// TIA Portal V19 export
FUNCTION_BLOCK "Area02_SafetyInterface_FB"   // FB207, LAD
TITLE = AREA 01 SAFETY INTERFACE
// stored: Access Published, MemoryReserve 100, SetENOAutomatically false
   VAR_INPUT
      AreaInterface : "AreaInterface";
      Passivation : Bool;
   END_VAR
   VAR_OUTPUT
      MachineInterface : "MachineInterface";
      COut : Struct
         WarningsPresence : Bool;
         AlarmsPresence : Bool;
         PathTestRollformer_DriveCtrlSafe : Bool;
      END_STRUCT;
   END_VAR
   VAR_IN_OUT
      Alarm : Struct
         FDBACK_Error : Struct
            F_Contactor_Rollformer_CambioFormato : Bool;
            F_Contactor_FinalCut_HU_Motor : Bool;
            F_Contactor_FinalCut_HU_Valve : Bool;
         END_STRUCT;
         S120_SafetyFaultActive : Struct
            Cassetta1_OP : Bool;
            Cassetta1_MOT : Bool;
            Cassetta2_OP : Bool;
            Cassetta2_MOT : Bool;
            Cassetta3_OP : Bool;
            Cassetta3_MOT : Bool;
            Rollformer : Bool;
            FAK_PusherAx : Bool;
            FlyCarriage : Bool;
            AccRolls1 : Bool;
            AccRolls2 : Bool;
            AccRolls3 : Bool;
         END_STRUCT;
         UnathorizedOpen : Struct
            D10 : Bool;
            D11 : Bool;
            D12 : Bool;
            D14 : Bool;
            D15 : Bool;
            D16 : Bool;
            D18 : Bool;
         END_STRUCT;
         PathTest_Rollformer : Bool;
      END_STRUCT;
      Warning : Struct
         Selectors : Struct
            Maintenance_MB2 : Bool;
         END_STRUCT;
         Feedback : Struct
            F_Valve_Area02_HU : Bool;
         END_STRUCT;
         DoorOpened : Struct
            D10 : Bool;
            D11 : Bool;
            D12 : Bool;
            D14 : Bool;
            D15 : Bool;
            D16 : Bool;
            D18 : Bool;
         END_STRUCT;
         DoorOpenRequest : Struct
            D10 : Bool;
            D11 : Bool;
            D12 : Bool;
            D14 : Bool;
            D15 : Bool;
            D16 : Bool;
            D18 : Bool;
         END_STRUCT;
         PathTest_Rollformer : Bool;
      END_STRUCT;
   END_VAR
   VAR
      Sts : Struct
         FdbackErrorPresence : Bool;
         S120SftyFaultPresence : Bool;
         DoorUnauthorizedOpen : Bool;
         DoorOpened { ExternalAccessible := 'False'; ExternalVisible := 'False'; ExternalWritable := 'False'} : Bool;
         DoorOpenRequest : Bool;
         DoorNotLocked : Bool;
      END_STRUCT;
      PathTest_Rollformer { S7_SetPoint := 'True'} : "PathTest";
   END_VAR
   VAR_TEMP
      SteadyOn : Bool;
      BlinkFast : Bool;
      BlinkLow : Bool;
      DummyLamp : Bool;
   END_VAR
BEGIN

REGION Network 1: <<<< C O N T R O L S A F E T Y D I A G N O S T I C >>>>>
END_REGION

REGION Network 2 (SCL): Fdback error


   #Alarm.FDBACK_Error.F_Contactor_Rollformer_CambioFormato := "Main_Safety_RTG1_DB".F_Zone11.F_Contactor_CambioFormato_Profilatrice.ERROR;
   #Alarm.FDBACK_Error.F_Contactor_FinalCut_HU_Motor := "Main_Safety_RTG1_DB".F_Zone13.F_Contactor_HU_FinalCut_Motor.ERROR;
   #Alarm.FDBACK_Error.F_Contactor_FinalCut_HU_Valve := "Main_Safety_RTG1_DB".F_Zone13.F_SafetyValve_FinalCut.FDO_FBK_ERROR;
END_REGION

REGION Network 3 (SCL): S120 Safety Fault

   #Alarm.S120_SafetyFaultActive.Cassetta1_OP := "Main_Safety_RTG1_DB".F_Zone11.F_Sinamics_Cassetta1_OP.SftyFault;
   #Alarm.S120_SafetyFaultActive.Cassetta1_MOT := "Main_Safety_RTG1_DB".F_Zone11.F_Sinamics_Cassetta1_MOT.SftyFault;
   #Alarm.S120_SafetyFaultActive.Cassetta2_OP := "Main_Safety_RTG1_DB".F_Zone11.F_Sinamics_Cassetta2_OP.SftyFault;
   #Alarm.S120_SafetyFaultActive.Cassetta2_MOT := "Main_Safety_RTG1_DB".F_Zone11.F_Sinamics_Cassetta2_MOT.SftyFault;
   #Alarm.S120_SafetyFaultActive.Cassetta3_OP := "Main_Safety_RTG1_DB".F_Zone11.F_Sinamics_Cassetta3_OP.SftyFault;
   #Alarm.S120_SafetyFaultActive.Cassetta3_MOT := "Main_Safety_RTG1_DB".F_Zone11.F_Sinamics_Cassetta3_MOT.SftyFault;
   #Alarm.S120_SafetyFaultActive.Rollformer := "Main_Safety_RTG1_DB".F_Zone20.F_Sinamics_Rollformer.SftyFault;
   #Alarm.S120_SafetyFaultActive.FAK_PusherAx := "Main_Safety_RTG1_DB".F_Zone13.F_Sinamics_FAK_Pusher.SftyFault;
   #Alarm.S120_SafetyFaultActive.FlyCarriage := "Main_Safety_RTG1_DB".F_Zone13.F_Sinamics_Carriage.SftyFault;
   #Alarm.S120_SafetyFaultActive.AccRolls1 := "Main_Safety_RTG1_DB".F_Zone15.F_Sinamics_AccRolls1.SftyFault;
   #Alarm.S120_SafetyFaultActive.AccRolls2 := "Main_Safety_RTG1_DB".F_Zone15.F_Sinamics_AccRolls2.SftyFault;
   #Alarm.S120_SafetyFaultActive.AccRolls3 := "Main_Safety_RTG1_DB".F_Zone15.F_Sinamics_AccRolls3.SftyFault;
END_REGION

REGION Network 4: Door D10 - Alarm unauthorized door opening
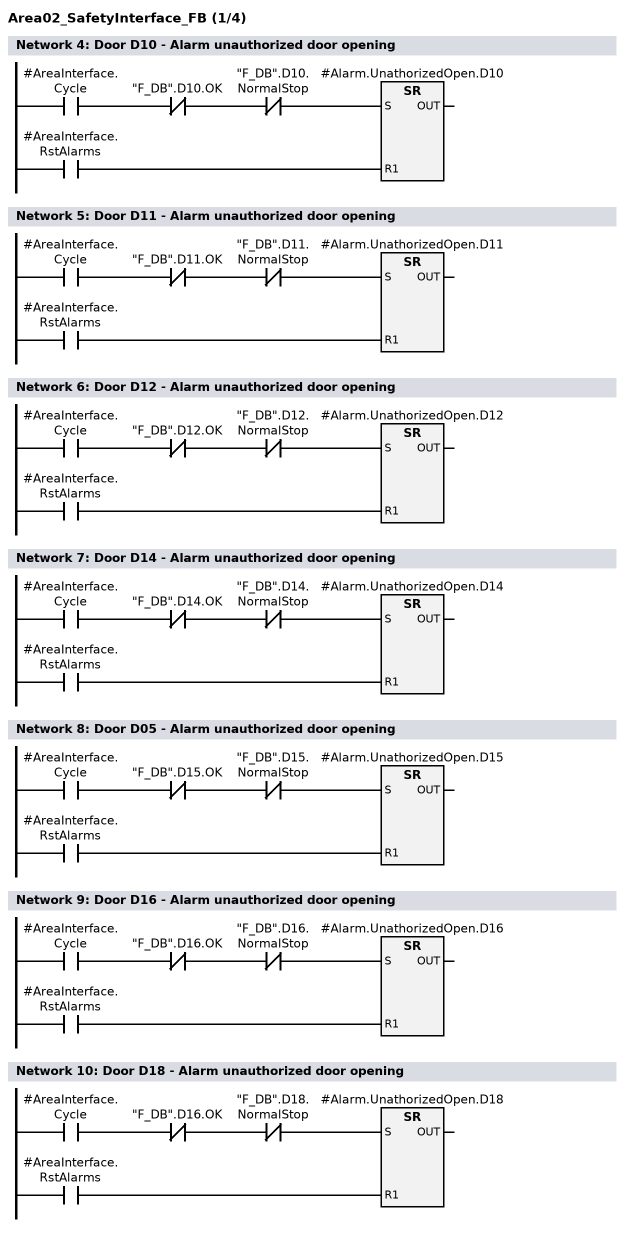
   RUNG wire#powerrail
      Contact( #AreaInterface.Cycle )
      I_Contact( "F_DB".D10.OK )
      I_Contact( "F_DB".D10.NormalStop )
      S_SR(operand := #Alarm.UnathorizedOpen.D10, r1 := wire#w1)
   END_RUNG
   RUNG wire#powerrail
      Contact( #AreaInterface.RstAlarms )
   END_RUNG wire#w1
   // the same network as SCL:
   IF #AreaInterface.Cycle AND NOT "F_DB".D10.OK AND NOT "F_DB".D10.NormalStop THEN
       #Alarm.UnathorizedOpen.D10 := TRUE;   // SR flip-flop
   END_IF;
   IF #AreaInterface.RstAlarms THEN #Alarm.UnathorizedOpen.D10 := FALSE; END_IF;
END_REGION

REGION Network 5: Door D11 - Alarm unauthorized door opening
   RUNG wire#powerrail
      Contact( #AreaInterface.Cycle )
      I_Contact( "F_DB".D11.OK )
      I_Contact( "F_DB".D11.NormalStop )
      S_SR(operand := #Alarm.UnathorizedOpen.D11, r1 := wire#w1)
   END_RUNG
   RUNG wire#powerrail
      Contact( #AreaInterface.RstAlarms )
   END_RUNG wire#w1
   // the same network as SCL:
   IF #AreaInterface.Cycle AND NOT "F_DB".D11.OK AND NOT "F_DB".D11.NormalStop THEN
       #Alarm.UnathorizedOpen.D11 := TRUE;   // SR flip-flop
   END_IF;
   IF #AreaInterface.RstAlarms THEN #Alarm.UnathorizedOpen.D11 := FALSE; END_IF;
END_REGION

REGION Network 6: Door D12 - Alarm unauthorized door opening
   RUNG wire#powerrail
      Contact( #AreaInterface.Cycle )
      I_Contact( "F_DB".D12.OK )
      I_Contact( "F_DB".D12.NormalStop )
      S_SR(operand := #Alarm.UnathorizedOpen.D12, r1 := wire#w1)
   END_RUNG
   RUNG wire#powerrail
      Contact( #AreaInterface.RstAlarms )
   END_RUNG wire#w1
   // the same network as SCL:
   IF #AreaInterface.Cycle AND NOT "F_DB".D12.OK AND NOT "F_DB".D12.NormalStop THEN
       #Alarm.UnathorizedOpen.D12 := TRUE;   // SR flip-flop
   END_IF;
   IF #AreaInterface.RstAlarms THEN #Alarm.UnathorizedOpen.D12 := FALSE; END_IF;
END_REGION

REGION Network 7: Door D14 - Alarm unauthorized door opening
   RUNG wire#powerrail
      Contact( #AreaInterface.Cycle )
      I_Contact( "F_DB".D14.OK )
      I_Contact( "F_DB".D14.NormalStop )
      S_SR(operand := #Alarm.UnathorizedOpen.D14, r1 := wire#w1)
   END_RUNG
   RUNG wire#powerrail
      Contact( #AreaInterface.RstAlarms )
   END_RUNG wire#w1
   // the same network as SCL:
   IF #AreaInterface.Cycle AND NOT "F_DB".D14.OK AND NOT "F_DB".D14.NormalStop THEN
       #Alarm.UnathorizedOpen.D14 := TRUE;   // SR flip-flop
   END_IF;
   IF #AreaInterface.RstAlarms THEN #Alarm.UnathorizedOpen.D14 := FALSE; END_IF;
END_REGION

REGION Network 8: Door D05 - Alarm unauthorized door opening
   RUNG wire#powerrail
      Contact( #AreaInterface.Cycle )
      I_Contact( "F_DB".D15.OK )
      I_Contact( "F_DB".D15.NormalStop )
      S_SR(operand := #Alarm.UnathorizedOpen.D15, r1 := wire#w1)
   END_RUNG
   RUNG wire#powerrail
      Contact( #AreaInterface.RstAlarms )
   END_RUNG wire#w1
   // the same network as SCL:
   IF #AreaInterface.Cycle AND NOT "F_DB".D15.OK AND NOT "F_DB".D15.NormalStop THEN
       #Alarm.UnathorizedOpen.D15 := TRUE;   // SR flip-flop
   END_IF;
   IF #AreaInterface.RstAlarms THEN #Alarm.UnathorizedOpen.D15 := FALSE; END_IF;
END_REGION

REGION Network 9: Door D16 - Alarm unauthorized door opening
   RUNG wire#powerrail
      Contact( #AreaInterface.Cycle )
      I_Contact( "F_DB".D16.OK )
      I_Contact( "F_DB".D16.NormalStop )
      S_SR(operand := #Alarm.UnathorizedOpen.D16, r1 := wire#w1)
   END_RUNG
   RUNG wire#powerrail
      Contact( #AreaInterface.RstAlarms )
   END_RUNG wire#w1
   // the same network as SCL:
   IF #AreaInterface.Cycle AND NOT "F_DB".D16.OK AND NOT "F_DB".D16.NormalStop THEN
       #Alarm.UnathorizedOpen.D16 := TRUE;   // SR flip-flop
   END_IF;
   IF #AreaInterface.RstAlarms THEN #Alarm.UnathorizedOpen.D16 := FALSE; END_IF;
END_REGION

REGION Network 10: Door D18 - Alarm unauthorized door opening
   RUNG wire#powerrail
      Contact( #AreaInterface.Cycle )
      I_Contact( "F_DB".D16.OK )
      I_Contact( "F_DB".D18.NormalStop )
      S_SR(operand := #Alarm.UnathorizedOpen.D18, r1 := wire#w1)
   END_RUNG
   RUNG wire#powerrail
      Contact( #AreaInterface.RstAlarms )
   END_RUNG wire#w1
   // the same network as SCL:
   IF #AreaInterface.Cycle AND NOT "F_DB".D16.OK AND NOT "F_DB".D18.NormalStop THEN
       #Alarm.UnathorizedOpen.D18 := TRUE;   // SR flip-flop
   END_IF;
   IF #AreaInterface.RstAlarms THEN #Alarm.UnathorizedOpen.D18 := FALSE; END_IF;
END_REGION

REGION Network 11: +
END_REGION

REGION Network 12: +
END_REGION

REGION Network 13: +
END_REGION

REGION Network 14: < < < < WARNINGS > > > >
END_REGION

REGION Network 15: Warning selector set-up MB2
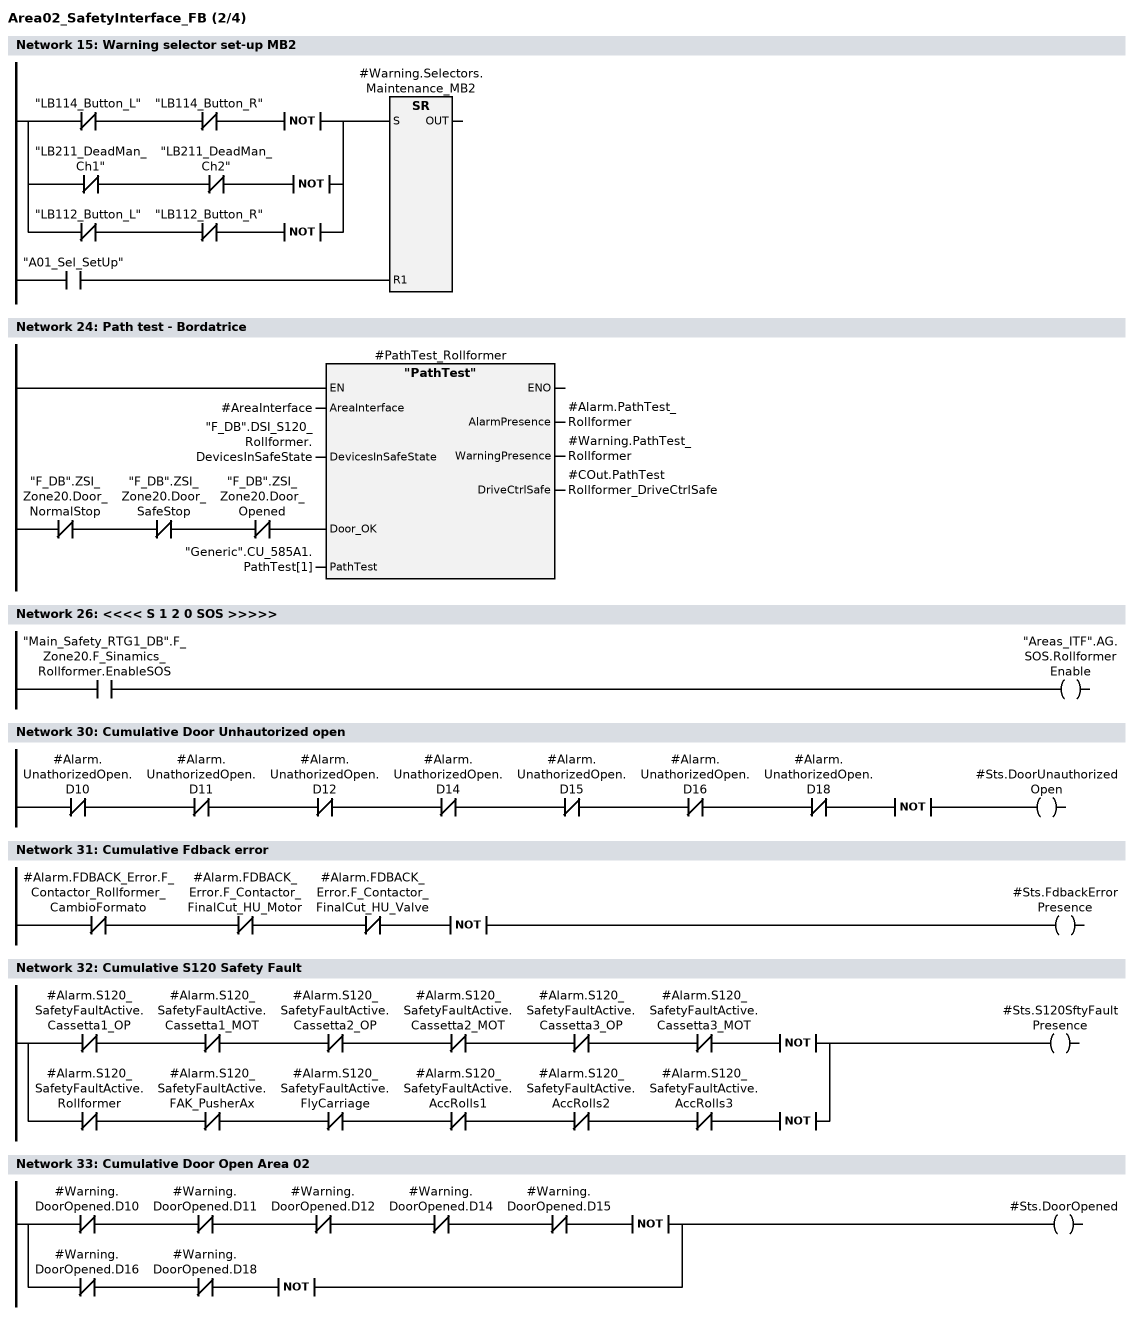
   RUNG wire#powerrail
      I_Contact( "LB114_Button_L" )
      I_Contact( "LB114_Button_R" )
      Not()
      wire#w1
      S_SR(operand := #Warning.Selectors.Maintenance_MB2, r1 := wire#w2)
   END_RUNG
   RUNG wire#powerrail
      I_Contact( "LB211_DeadMan_Ch1" )
      I_Contact( "LB211_DeadMan_Ch2" )
      Not()
   END_RUNG wire#w1
   RUNG wire#powerrail
      I_Contact( "LB112_Button_L" )
      I_Contact( "LB112_Button_R" )
      Not()
   END_RUNG wire#w1
   RUNG wire#powerrail
      Contact( "A01_Sel_SetUp" )
   END_RUNG wire#w2
   // the same network as SCL:
   IF NOT (NOT "LB114_Button_L" AND NOT "LB114_Button_R") OR NOT (NOT "LB211_DeadMan_Ch1" AND NOT "LB211_DeadMan_Ch2") OR NOT (NOT "LB112_Button_L" AND NOT "LB112_Button_R") THEN
       #Warning.Selectors.Maintenance_MB2 := TRUE;   // SR flip-flop
   END_IF;
   IF "A01_Sel_SetUp" THEN #Warning.Selectors.Maintenance_MB2 := FALSE; END_IF;
END_REGION

REGION Network 16 (SCL): Feddback valve

   #Warning.Feedback.F_Valve_Area02_HU := "Main_Safety_RTG1_DB".F_Zone13.F_SafetyValve_FinalCut.EV_SAFETY_FBK_WARNING;
END_REGION

REGION Network 17 (SCL): Door open
   //Door opened
   #Warning.DoorOpened.D10 := "F_DB".D10.Warning_DoorOpened;
   #Warning.DoorOpened.D11 := "F_DB".D11.Warning_DoorOpened;
   #Warning.DoorOpened.D12 := "F_DB".D12.Warning_DoorOpened;
   #Warning.DoorOpened.D14 := "F_DB".D14.Warning_DoorOpened;
   #Warning.DoorOpened.D15 := "F_DB".D15.Warning_DoorOpened;
   #Warning.DoorOpened.D16 := "F_DB".D16.Warning_DoorOpened;
   #Warning.DoorOpened.D18 := "F_DB".D18.Warning_DoorOpened;
END_REGION

REGION Network 18 (SCL): Door open request

   //Door open reequest
   #Warning.DoorOpenRequest.D10 := "F_DB".D10.Warning_DoorOpenRequest;
   #Warning.DoorOpenRequest.D11 := "F_DB".D11.Warning_DoorOpenRequest;
   #Warning.DoorOpenRequest.D12 := "F_DB".D12.Warning_DoorOpenRequest;
   #Warning.DoorOpenRequest.D14 := "F_DB".D14.Warning_DoorOpenRequest;
   #Warning.DoorOpenRequest.D15 := "F_DB".D15.Warning_DoorOpenRequest;
   #Warning.DoorOpenRequest.D16 := "F_DB".D16.Warning_DoorOpenRequest;
   #Warning.DoorOpenRequest.D18 := "F_DB".D18.Warning_DoorOpenRequest;
END_REGION

REGION Network 19 (SCL): Door not closed

   (*

   #Warning.DoorNotLocked.D04 := "D04_LockEnable" AND NOT "D04_Cancello_Bloccato";
   #Warning.DoorNotLocked.D05 := "D05_LockEnable" AND NOT "D05_Cancello_Bloccato";
   #Warning.DoorNotLocked.D07 := "D07_LockEnable" AND NOT "D07_Cancello_Bloccato";

   *)
END_REGION

REGION Network 20: +
END_REGION

REGION Network 21: +
END_REGION

REGION Network 22: +
END_REGION

REGION Network 23: <<<< S 1 2 0 D R I V E P A T H T E S T >>>>>
END_REGION

REGION Network 24: Path test - Bordatrice
   RUNG wire#powerrail
      #PathTest_Rollformer(Door_OK := wire#w1, AreaInterface := #AreaInterface, DevicesInSafeState := "F_DB".DSI_S120_Rollformer.DevicesInSafeState, PathTest := "Generic".CU_585A1.PathTest[1], AlarmPresence => #Alarm.PathTest_Rollformer, WarningPresence => #Warning.PathTest_Rollformer, DriveCtrlSafe => #COut.PathTestRollformer_DriveCtrlSafe)
   END_RUNG
   RUNG wire#powerrail
      I_Contact( "F_DB".ZSI_Zone20.Door_NormalStop )
      I_Contact( "F_DB".ZSI_Zone20.Door_SafeStop )
      I_Contact( "F_DB".ZSI_Zone20.Door_Opened )
   END_RUNG wire#w1
   // the same network as SCL:
   #PathTest_Rollformer(AreaInterface := #AreaInterface,   // "PathTest"
                        DevicesInSafeState := "F_DB".DSI_S120_Rollformer.DevicesInSafeState,
                        Door_OK := NOT "F_DB".ZSI_Zone20.Door_NormalStop AND NOT "F_DB".ZSI_Zone20.Door_SafeStop AND NOT "F_DB".ZSI_Zone20.Door_Opened,
                        PathTest := "Generic".CU_585A1.PathTest[1],
                        AlarmPresence => #Alarm.PathTest_Rollformer,
                        WarningPresence => #Warning.PathTest_Rollformer,
                        DriveCtrlSafe => #COut.PathTestRollformer_DriveCtrlSafe);
END_REGION

REGION Network 25: +
END_REGION

REGION Network 26: <<<< S 1 2 0 SOS >>>>>
   RUNG wire#powerrail
      Contact( "Main_Safety_RTG1_DB".F_Zone20.F_Sinamics_Rollformer.EnableSOS )
      Coil( "Areas_ITF".AG.SOS.RollformerEnable )
   END_RUNG
   // the same network as SCL:
   "Areas_ITF".AG.SOS.RollformerEnable := "Main_Safety_RTG1_DB".F_Zone20.F_Sinamics_Rollformer.EnableSOS;
END_REGION

REGION Network 27: +
END_REGION

REGION Network 28: +
END_REGION

REGION Network 29: < < < < C U M U L A T I V E > > > >
END_REGION

REGION Network 30: Cumulative Door Unhautorized open
   RUNG wire#powerrail
      I_Contact( #Alarm.UnathorizedOpen.D10 )
      I_Contact( #Alarm.UnathorizedOpen.D11 )
      I_Contact( #Alarm.UnathorizedOpen.D12 )
      I_Contact( #Alarm.UnathorizedOpen.D14 )
      I_Contact( #Alarm.UnathorizedOpen.D15 )
      I_Contact( #Alarm.UnathorizedOpen.D16 )
      I_Contact( #Alarm.UnathorizedOpen.D18 )
      Not()
      Coil( #Sts.DoorUnauthorizedOpen )
   END_RUNG
   // the same network as SCL:
   #Sts.DoorUnauthorizedOpen := NOT (NOT #Alarm.UnathorizedOpen.D10 AND NOT #Alarm.UnathorizedOpen.D11 AND NOT #Alarm.UnathorizedOpen.D12 AND NOT #Alarm.UnathorizedOpen.D14 AND NOT #Alarm.UnathorizedOpen.D15 AND NOT #Alarm.UnathorizedOpen.D16 AND NOT #Alarm.UnathorizedOpen.D18);
END_REGION

REGION Network 31: Cumulative Fdback error
   RUNG wire#powerrail
      I_Contact( #Alarm.FDBACK_Error.F_Contactor_Rollformer_CambioFormato )
      I_Contact( #Alarm.FDBACK_Error.F_Contactor_FinalCut_HU_Motor )
      I_Contact( #Alarm.FDBACK_Error.F_Contactor_FinalCut_HU_Valve )
      Not()
      Coil( #Sts.FdbackErrorPresence )
   END_RUNG
   // the same network as SCL:
   #Sts.FdbackErrorPresence := NOT (NOT #Alarm.FDBACK_Error.F_Contactor_Rollformer_CambioFormato AND NOT #Alarm.FDBACK_Error.F_Contactor_FinalCut_HU_Motor AND NOT #Alarm.FDBACK_Error.F_Contactor_FinalCut_HU_Valve);
END_REGION

REGION Network 32: Cumulative S120 Safety Fault
   RUNG wire#powerrail
      I_Contact( #Alarm.S120_SafetyFaultActive.Cassetta1_OP )
      I_Contact( #Alarm.S120_SafetyFaultActive.Cassetta1_MOT )
      I_Contact( #Alarm.S120_SafetyFaultActive.Cassetta2_OP )
      I_Contact( #Alarm.S120_SafetyFaultActive.Cassetta2_MOT )
      I_Contact( #Alarm.S120_SafetyFaultActive.Cassetta3_OP )
      I_Contact( #Alarm.S120_SafetyFaultActive.Cassetta3_MOT )
      Not()
      wire#w1
      Coil( #Sts.S120SftyFaultPresence )
   END_RUNG
   RUNG wire#powerrail
      I_Contact( #Alarm.S120_SafetyFaultActive.Rollformer )
      I_Contact( #Alarm.S120_SafetyFaultActive.FAK_PusherAx )
      I_Contact( #Alarm.S120_SafetyFaultActive.FlyCarriage )
      I_Contact( #Alarm.S120_SafetyFaultActive.AccRolls1 )
      I_Contact( #Alarm.S120_SafetyFaultActive.AccRolls2 )
      I_Contact( #Alarm.S120_SafetyFaultActive.AccRolls3 )
      Not()
   END_RUNG wire#w1
   // the same network as SCL:
   #Sts.S120SftyFaultPresence := NOT (NOT #Alarm.S120_SafetyFaultActive.Cassetta1_OP AND NOT #Alarm.S120_SafetyFaultActive.Cassetta1_MOT AND NOT #Alarm.S120_SafetyFaultActive.Cassetta2_OP AND NOT #Alarm.S120_SafetyFaultActive.Cassetta2_MOT AND NOT #Alarm.S120_SafetyFaultActive.Cassetta3_OP AND NOT #Alarm.S120_SafetyFaultActive.Cassetta3_MOT) OR NOT (NOT #Alarm.S120_SafetyFaultActive.Rollformer AND NOT #Alarm.S120_SafetyFaultActive.FAK_PusherAx AND NOT #Alarm.S120_SafetyFaultActive.FlyCarriage AND NOT #Alarm.S120_SafetyFaultActive.AccRolls1 AND NOT #Alarm.S120_SafetyFaultActive.AccRolls2 AND NOT #Alarm.S120_SafetyFaultActive.AccRolls3);
END_REGION

REGION Network 33: Cumulative Door Open Area 02
   RUNG wire#powerrail
      I_Contact( #Warning.DoorOpened.D10 )
      I_Contact( #Warning.DoorOpened.D11 )
      I_Contact( #Warning.DoorOpened.D12 )
      I_Contact( #Warning.DoorOpened.D14 )
      I_Contact( #Warning.DoorOpened.D15 )
      Not()
      wire#w1
      Coil( #Sts.DoorOpened )
   END_RUNG
   RUNG wire#powerrail
      I_Contact( #Warning.DoorOpened.D16 )
      I_Contact( #Warning.DoorOpened.D18 )
      Not()
   END_RUNG wire#w1
   // the same network as SCL:
   #Sts.DoorOpened := NOT (NOT #Warning.DoorOpened.D10 AND NOT #Warning.DoorOpened.D11 AND NOT #Warning.DoorOpened.D12 AND NOT #Warning.DoorOpened.D14 AND NOT #Warning.DoorOpened.D15) OR NOT (NOT #Warning.DoorOpened.D16 AND NOT #Warning.DoorOpened.D18);
END_REGION

REGION Network 34: Cumulative Door Open Request Area
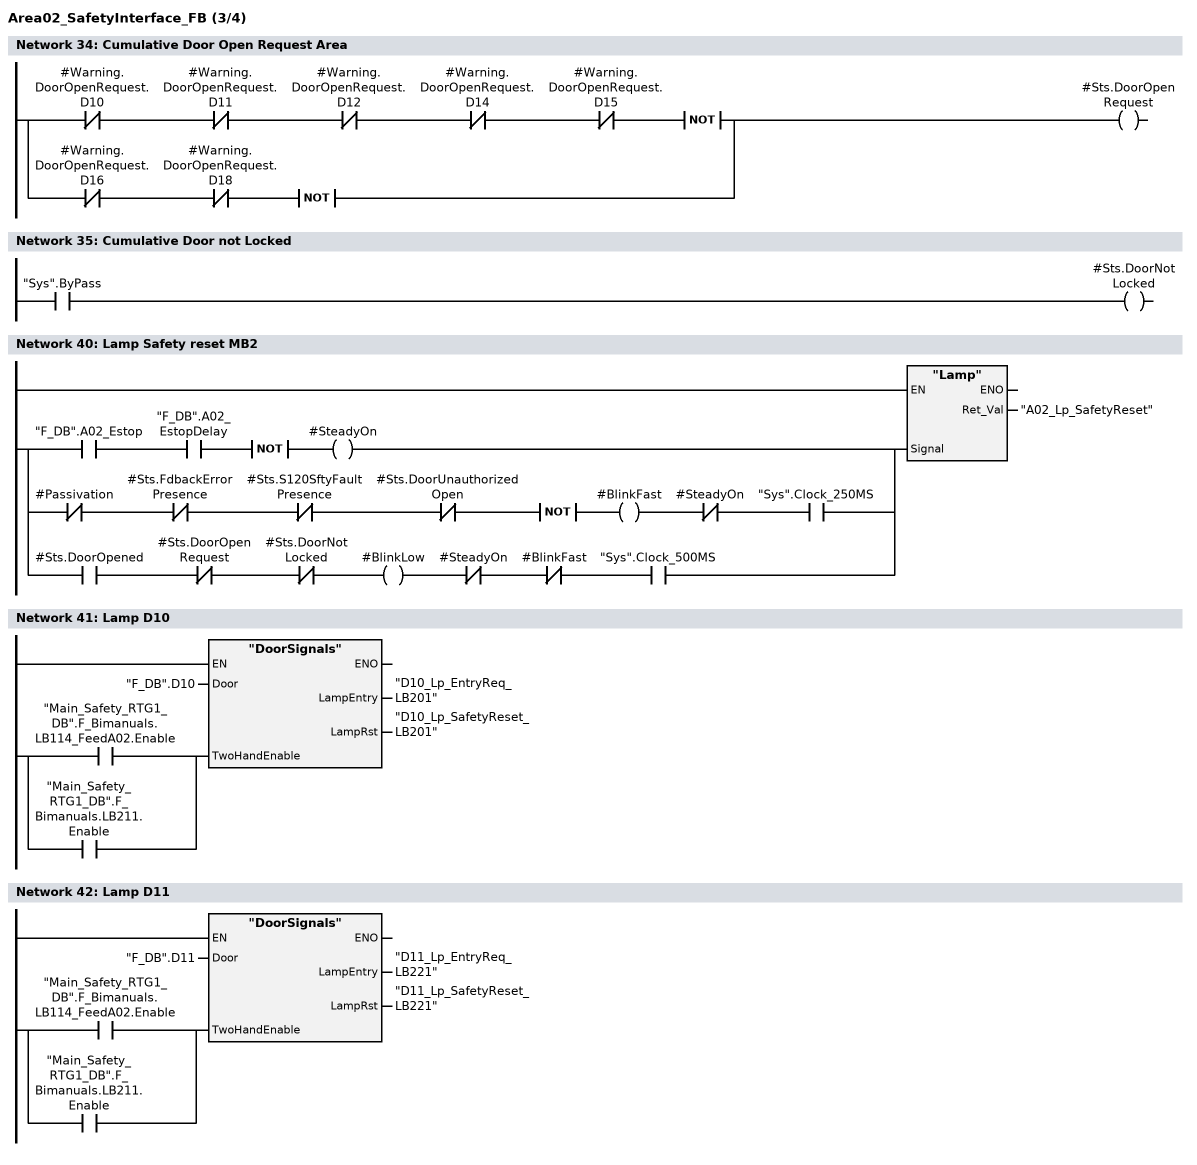
   RUNG wire#powerrail
      I_Contact( #Warning.DoorOpenRequest.D10 )
      I_Contact( #Warning.DoorOpenRequest.D11 )
      I_Contact( #Warning.DoorOpenRequest.D12 )
      I_Contact( #Warning.DoorOpenRequest.D14 )
      I_Contact( #Warning.DoorOpenRequest.D15 )
      Not()
      wire#w1
      Coil( #Sts.DoorOpenRequest )
   END_RUNG
   RUNG wire#powerrail
      I_Contact( #Warning.DoorOpenRequest.D16 )
      I_Contact( #Warning.DoorOpenRequest.D18 )
      Not()
   END_RUNG wire#w1
   // the same network as SCL:
   #Sts.DoorOpenRequest := NOT (NOT #Warning.DoorOpenRequest.D10 AND NOT #Warning.DoorOpenRequest.D11 AND NOT #Warning.DoorOpenRequest.D12 AND NOT #Warning.DoorOpenRequest.D14 AND NOT #Warning.DoorOpenRequest.D15) OR NOT (NOT #Warning.DoorOpenRequest.D16 AND NOT #Warning.DoorOpenRequest.D18);
END_REGION

REGION Network 35: Cumulative Door not Locked
   RUNG wire#powerrail
      Contact( "Sys".ByPass )
      Coil( #Sts.DoorNotLocked )
   END_RUNG
   // the same network as SCL:
   #Sts.DoorNotLocked := "Sys".ByPass;
END_REGION

REGION Network 36: +
END_REGION

REGION Network 37: +
END_REGION

REGION Network 38: +
END_REGION

REGION Network 39: < < < L A M P S > > >
END_REGION

REGION Network 40: Lamp Safety reset MB2
   RUNG wire#powerrail
      "Lamp"(Signal := wire#w1, Ret_Val => "A02_Lp_SafetyReset")
   END_RUNG
   RUNG wire#powerrail
      Contact( "F_DB".A02_Estop )
      Contact( "F_DB".A02_EstopDelay )
      Not()
      Coil( #SteadyOn )
   END_RUNG wire#w1
   RUNG wire#powerrail
      I_Contact( #Passivation )
      I_Contact( #Sts.FdbackErrorPresence )
      I_Contact( #Sts.S120SftyFaultPresence )
      I_Contact( #Sts.DoorUnauthorizedOpen )
      Not()
      Coil( #BlinkFast )
      I_Contact( #SteadyOn )
      Contact( "Sys".Clock_250MS )
   END_RUNG wire#w1
   RUNG wire#powerrail
      Contact( #Sts.DoorOpened )
      I_Contact( #Sts.DoorOpenRequest )
      I_Contact( #Sts.DoorNotLocked )
      Coil( #BlinkLow )
      I_Contact( #SteadyOn )
      I_Contact( #BlinkFast )
      Contact( "Sys".Clock_500MS )
   END_RUNG wire#w1
   // the same network as SCL:
   #SteadyOn := NOT ("F_DB".A02_Estop AND "F_DB".A02_EstopDelay);
   #BlinkFast := NOT (NOT #Passivation AND NOT #Sts.FdbackErrorPresence AND NOT #Sts.S120SftyFaultPresence AND NOT #Sts.DoorUnauthorizedOpen);
   #BlinkLow := #Sts.DoorOpened AND NOT #Sts.DoorOpenRequest AND NOT #Sts.DoorNotLocked;
   "A02_Lp_SafetyReset" := "Lamp"(Signal := #SteadyOn OR (#BlinkFast AND NOT #SteadyOn AND "Sys".Clock_250MS) OR (#BlinkLow AND NOT #SteadyOn AND NOT #BlinkFast AND "Sys".Clock_500MS));
END_REGION

REGION Network 41: Lamp D10
   RUNG wire#powerrail
      "DoorSignals"(TwoHandEnable := wire#w1, Door := "F_DB".D10, LampEntry => "D10_Lp_EntryReq_LB201", LampRst => "D10_Lp_SafetyReset_LB201")
   END_RUNG
   RUNG wire#powerrail
      Contact( "Main_Safety_RTG1_DB".F_Bimanuals.LB114_FeedA02.Enable )
   END_RUNG wire#w1
   RUNG wire#powerrail
      Contact( "Main_Safety_RTG1_DB".F_Bimanuals.LB211.Enable )
   END_RUNG wire#w1
   // the same network as SCL:
   "DoorSignals"(Door := "F_DB".D10,
                 TwoHandEnable := "Main_Safety_RTG1_DB".F_Bimanuals.LB114_FeedA02.Enable OR "Main_Safety_RTG1_DB".F_Bimanuals.LB211.Enable,
                 LampEntry => "D10_Lp_EntryReq_LB201",
                 LampRst => "D10_Lp_SafetyReset_LB201");
END_REGION

REGION Network 42: Lamp D11
   RUNG wire#powerrail
      "DoorSignals"(TwoHandEnable := wire#w1, Door := "F_DB".D11, LampEntry => "D11_Lp_EntryReq_LB221", LampRst => "D11_Lp_SafetyReset_LB221")
   END_RUNG
   RUNG wire#powerrail
      Contact( "Main_Safety_RTG1_DB".F_Bimanuals.LB114_FeedA02.Enable )
   END_RUNG wire#w1
   RUNG wire#powerrail
      Contact( "Main_Safety_RTG1_DB".F_Bimanuals.LB211.Enable )
   END_RUNG wire#w1
   // the same network as SCL:
   "DoorSignals"(Door := "F_DB".D11,
                 TwoHandEnable := "Main_Safety_RTG1_DB".F_Bimanuals.LB114_FeedA02.Enable OR "Main_Safety_RTG1_DB".F_Bimanuals.LB211.Enable,
                 LampEntry => "D11_Lp_EntryReq_LB221",
                 LampRst => "D11_Lp_SafetyReset_LB221");
END_REGION

REGION Network 43: Lamp D12
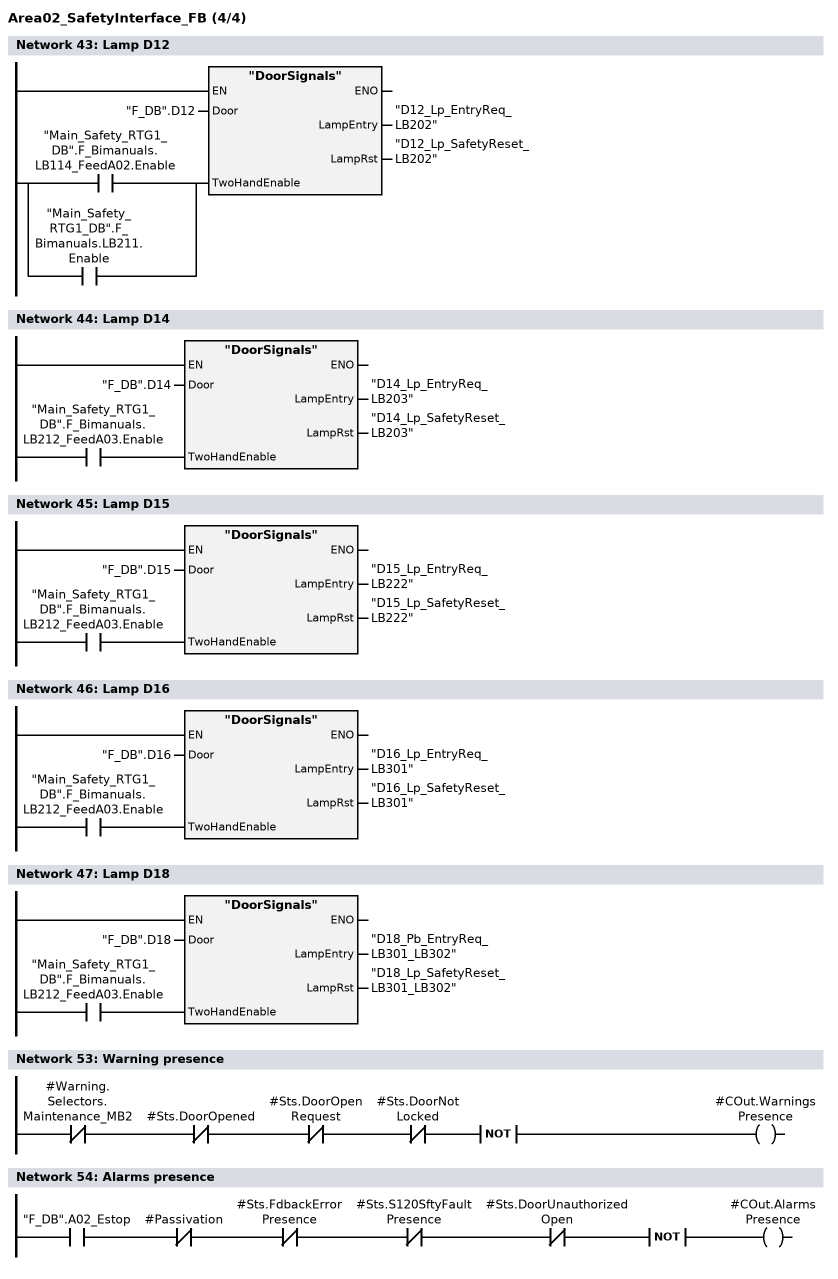
   RUNG wire#powerrail
      "DoorSignals"(TwoHandEnable := wire#w1, Door := "F_DB".D12, LampEntry => "D12_Lp_EntryReq_LB202", LampRst => "D12_Lp_SafetyReset_LB202")
   END_RUNG
   RUNG wire#powerrail
      Contact( "Main_Safety_RTG1_DB".F_Bimanuals.LB114_FeedA02.Enable )
   END_RUNG wire#w1
   RUNG wire#powerrail
      Contact( "Main_Safety_RTG1_DB".F_Bimanuals.LB211.Enable )
   END_RUNG wire#w1
   // the same network as SCL:
   "DoorSignals"(Door := "F_DB".D12,
                 TwoHandEnable := "Main_Safety_RTG1_DB".F_Bimanuals.LB114_FeedA02.Enable OR "Main_Safety_RTG1_DB".F_Bimanuals.LB211.Enable,
                 LampEntry => "D12_Lp_EntryReq_LB202",
                 LampRst => "D12_Lp_SafetyReset_LB202");
END_REGION

REGION Network 44: Lamp D14
   RUNG wire#powerrail
      "DoorSignals"(TwoHandEnable := wire#w1, Door := "F_DB".D14, LampEntry => "D14_Lp_EntryReq_LB203", LampRst => "D14_Lp_SafetyReset_LB203")
   END_RUNG
   RUNG wire#powerrail
      Contact( "Main_Safety_RTG1_DB".F_Bimanuals.LB212_FeedA03.Enable )
   END_RUNG wire#w1
   // the same network as SCL:
   "DoorSignals"(Door := "F_DB".D14,
                 TwoHandEnable := "Main_Safety_RTG1_DB".F_Bimanuals.LB212_FeedA03.Enable,
                 LampEntry => "D14_Lp_EntryReq_LB203",
                 LampRst => "D14_Lp_SafetyReset_LB203");
END_REGION

REGION Network 45: Lamp D15
   RUNG wire#powerrail
      "DoorSignals"(TwoHandEnable := wire#w1, Door := "F_DB".D15, LampEntry => "D15_Lp_EntryReq_LB222", LampRst => "D15_Lp_SafetyReset_LB222")
   END_RUNG
   RUNG wire#powerrail
      Contact( "Main_Safety_RTG1_DB".F_Bimanuals.LB212_FeedA03.Enable )
   END_RUNG wire#w1
   // the same network as SCL:
   "DoorSignals"(Door := "F_DB".D15,
                 TwoHandEnable := "Main_Safety_RTG1_DB".F_Bimanuals.LB212_FeedA03.Enable,
                 LampEntry => "D15_Lp_EntryReq_LB222",
                 LampRst => "D15_Lp_SafetyReset_LB222");
END_REGION

REGION Network 46: Lamp D16
   RUNG wire#powerrail
      "DoorSignals"(TwoHandEnable := wire#w1, Door := "F_DB".D16, LampEntry => "D16_Lp_EntryReq_LB301", LampRst => "D16_Lp_SafetyReset_LB301")
   END_RUNG
   RUNG wire#powerrail
      Contact( "Main_Safety_RTG1_DB".F_Bimanuals.LB212_FeedA03.Enable )
   END_RUNG wire#w1
   // the same network as SCL:
   "DoorSignals"(Door := "F_DB".D16,
                 TwoHandEnable := "Main_Safety_RTG1_DB".F_Bimanuals.LB212_FeedA03.Enable,
                 LampEntry => "D16_Lp_EntryReq_LB301",
                 LampRst => "D16_Lp_SafetyReset_LB301");
END_REGION

REGION Network 47: Lamp D18
   RUNG wire#powerrail
      "DoorSignals"(TwoHandEnable := wire#w1, Door := "F_DB".D18, LampEntry => "D18_Pb_EntryReq_LB301_LB302", LampRst => "D18_Lp_SafetyReset_LB301_LB302")
   END_RUNG
   RUNG wire#powerrail
      Contact( "Main_Safety_RTG1_DB".F_Bimanuals.LB212_FeedA03.Enable )
   END_RUNG wire#w1
   // the same network as SCL:
   "DoorSignals"(Door := "F_DB".D18,
                 TwoHandEnable := "Main_Safety_RTG1_DB".F_Bimanuals.LB212_FeedA03.Enable,
                 LampEntry => "D18_Pb_EntryReq_LB301_LB302",
                 LampRst => "D18_Lp_SafetyReset_LB301_LB302");
END_REGION

REGION Network 48: +
END_REGION

REGION Network 49: +
END_REGION

REGION Network 50: +
END_REGION

REGION Network 52: < < < < F I N A L > > > >
END_REGION

REGION Network 53: Warning presence
   RUNG wire#powerrail
      I_Contact( #Warning.Selectors.Maintenance_MB2 )
      I_Contact( #Sts.DoorOpened )
      I_Contact( #Sts.DoorOpenRequest )
      I_Contact( #Sts.DoorNotLocked )
      Not()
      Coil( #COut.WarningsPresence )
   END_RUNG
   // the same network as SCL:
   #COut.WarningsPresence := NOT (NOT #Warning.Selectors.Maintenance_MB2 AND NOT #Sts.DoorOpened AND NOT #Sts.DoorOpenRequest AND NOT #Sts.DoorNotLocked);
END_REGION

REGION Network 54: Alarms presence
   RUNG wire#powerrail
      Contact( "F_DB".A02_Estop )
      I_Contact( #Passivation )
      I_Contact( #Sts.FdbackErrorPresence )
      I_Contact( #Sts.S120SftyFaultPresence )
      I_Contact( #Sts.DoorUnauthorizedOpen )
      Not()
      Coil( #COut.AlarmsPresence )
   END_RUNG
   // the same network as SCL:
   #COut.AlarmsPresence := NOT ("F_DB".A02_Estop AND NOT #Passivation AND NOT #Sts.FdbackErrorPresence AND NOT #Sts.S120SftyFaultPresence AND NOT #Sts.DoorUnauthorizedOpen);
END_REGION

REGION Network 55: >
END_REGION

REGION Network 56: >
END_REGION

REGION Network 57 (SCL): Area ITF
   "Areas_ITF".A02.Doors_Closed :=
   NOT "F_DB".ZSI_Zone11.Door_Opened;
END_REGION

REGION Network 58: >
END_REGION

REGION Network 59 (SCL): Collect machine to zone interface

   #MachineInterface.AutReady := #AreaInterface.Aut AND NOT #COut.AlarmsPresence;
   #MachineInterface.Aborting := #COut.AlarmsPresence;
   #MachineInterface.MotionsStandStill := TRUE;
   #MachineInterface.AckStopInPhase := #AreaInterface.StopInPhase;
   #MachineInterface.AckStopProgrammed := #AreaInterface.StopProgrammed;
   #MachineInterface.AlarmsPresence := #COut.AlarmsPresence;
   #MachineInterface.WarningPresence := #COut.WarningsPresence;
END_REGION
END_FUNCTION_BLOCK
